LIN {X 0,Y 93.213,Z 295.861,A -85,B 0,C 180,E1 -28398.926,E2 -28398.926} C_VEL
LIN {X 0,Y 93.368,Z 291.962,A -85,B 0,C 180,E1 -28402.974,E2 -28402.974} C_VEL
LIN {X 0,Y 93.007,Z 287.711,A -85,B 0,C 180,E1 -28408.065,E2 -28408.065} C_VEL
LIN {X 0,Y 92.351,Z 284.316,A -85,B 0,C 180,E1 -28412.831,E2 -28412.831} C_VEL
LIN {X 0,Y 91.626,Z 281.752,A -85,B 0,C 180,E1 -28417.448,E2 -28417.448} C_VEL
LIN {X 0,Y 90.889,Z 279.975,A -85,B 0,C 180,E1 -28421.983,E2 -28421.983} C_VEL
LIN {X 0,Y 90.313,Z 278.726,A -85,B 0,C 180,E1 -28426.499,E2 -28426.499} C_VEL
LIN {X 0,Y 90.228,Z 277.226,A -85,B 0,C 180,E1 -28435.532,E2 -28435.532} C_VEL
LIN {X 0,Y 90.218,Z 278.004,A -85,B 0,C 180,E1 -28440,E2 -28440} C_VEL
LIN {X 0,Y 90.527,Z 282.078,A -85,B 0,C 180,E1 -28448.932,E2 -28448.932} C_VEL
LIN {X 0,Y 90.825,Z 283.273,A -85,B 0,C 180,E1 -28451.154,E2 -28451.154} C_VEL
LIN {X 0,Y 91.764,Z 288.136,A -85,B 0,C 180,E1 -28457.839,E2 -28457.839} C_VEL
LIN {X 0,Y 92.621,Z 293.238,A -85,B 0,C 180,E1 -28463.436,E2 -28463.436} C_VEL
LIN {X 0,Y 93.061,Z 299.729,A -85,B 0,C 180,E1 -28469.116,E2 -28469.116} C_VEL
LIN {X 0,Y 92.858,Z 301.798,A -85,B 0,C 180,E1 -28470.669,E2 -28470.669} C_VEL
LIN {X 0,Y 88.458,Z 309.904,A -85,B 0,C 180,E1 -28474.499,E2 -28474.499} C_VEL
LIN {X 0,Y 84.607,Z 315.889,A -85,B 0,C 180,E1 -28477.906,E2 -28477.906} C_VEL
LIN {X 0,Y 79.559,Z 323.019,A -85,B 0,C 180,E1 -28483.226,E2 -28483.226} C_VEL
LIN {X 0,Y 76.501,Z 327.119,A -85,B 0,C 180,E1 -28487.303,E2 -28487.303} C_VEL
LIN {X 0,Y 71.589,Z 332.386,A -85,B 0,C 180,E1 -28493.921,E2 -28493.921} C_VEL
LIN {X 0,Y 67.611,Z 336.755,A -85,B 0,C 180,E1 -28502.12,E2 -28502.12} C_VEL
LIN {X 0,Y 65.314,Z 339.861,A -85,B 0,C 180,E1 -28511.176,E2 -28511.176} C_VEL
LIN {X 0,Y 64.793,Z 341.313,A -85,B 0,C 180,E1 -28517.479,E2 -28517.479} C_VEL
LIN {X 0,Y 65.135,Z 342.235,A -85,B 0,C 180,E1 -28523.814,E2 -28523.814} C_VEL
LIN {X 0,Y 66.298,Z 342.706,A -85,B 0,C 180,E1 -28530.008,E2 -28530.008} C_VEL
LIN {X 0,Y 68.211,Z 342.64,A -85,B 0,C 180,E1 -28535.921,E2 -28535.921} C_VEL
LIN {X 0,Y 70.296,Z 342.047,A -85,B 0,C 180,E1 -28541.542,E2 -28541.542} C_VEL
LIN {X 0,Y 72.197,Z 340.793,A -85,B 0,C 180,E1 -28546.987,E2 -28546.987} C_VEL
LIN {X 0,Y 76.443,Z 338.002,A -85,B 0,C 180,E1 -28554.627,E2 -28554.627} C_VEL
LIN {X 0,Y 81.501,Z 346.039,A -85,B 0,C 180,E1 -28567.138,E2 -28567.138} C_VEL
LIN {X 0,Y 88.681,Z 351.555,A -85,B 0,C 180,E1 -28575.508,E2 -28575.508} C_VEL
LIN {X 0,Y 87.895,Z 350.817,A -85,B 0,C 180,E1 -28576.839,E2 -28576.839} C_VEL
LIN {X 0,Y 79.876,Z 342.499,A -85,B 0,C 180,E1 -28585.116,E2 -28585.116} C_VEL
LIN {X 0,Y 74.572,Z 333.187,A -85,B 0,C 180,E1 -28594.906,E2 -28594.906} C_VEL
LIN {X 0,Y 72.081,Z 324.848,A -85,B 0,C 180,E1 -28602.992,E2 -28602.992} C_VEL
LIN {X 0,Y 70.815,Z 316.559,A -85,B 0,C 180,E1 -28609.999,E2 -28609.999} C_VEL
LIN {X 0,Y 70.007,Z 307.489,A -85,B 0,C 180,E1 -28616.403,E2 -28616.403} C_VEL
LIN {X 0,Y 69.871,Z 305.556,A -85,B 0,C 180,E1 -28617.658,E2 -28617.658} C_VEL
LIN {X 0,Y 68.986,Z 305.923,A -85,B 0,C 180,E1 -28620,E2 -28620} C_VEL
LIN {X 0,Y 70.177,Z 304.044,A -85,B 0,C 180,E1 -28625.748,E2 -28625.748} C_VEL
LIN {X 0,Y 70.795,Z 303.378,A -85,B 0,C 180,E1 -28626.86,E2 -28626.86} C_VEL
LIN {X 0,Y 72.084,Z 302.243,A -85,B 0,C 180,E1 -28632.814,E2 -28632.814} C_VEL
LIN {X 0,Y 74.469,Z 300.381,A -85,B 0,C 180,E1 -28636.447,E2 -28636.447} C_VEL
LIN {X 0,Y 89.11,Z 292.891,A -85,B 0,C 180,E1 -28653.51,E2 -28653.51} C_VEL
LIN {X 0,Y 92.631,Z 292.592,A -85,B 0,C 180,E1 -28657.371,E2 -28657.371} C_VEL
LIN {X 0,Y 93.289,Z 293.19,A -85,B 0,C 180,E1 -28658.683,E2 -28658.683} C_VEL
LIN {X 0,Y 92.863,Z 296.646,A -85,B 0,C 180,E1 -28662.091,E2 -28662.091} C_VEL
LIN {X 0,Y 91.993,Z 299.53,A -85,B 0,C 180,E1 -28664.531,E2 -28664.531} C_VEL
LIN {X 0,Y 87.12,Z 305.638,A -85,B 0,C 180,E1 -28668.269,E2 -28668.269} C_VEL
LIN {X 0,Y 81.736,Z 311.304,A -85,B 0,C 180,E1 -28672.987,E2 -28672.987} C_VEL
LIN {X 0,Y 77.939,Z 314.962,A -85,B 0,C 180,E1 -28677.238,E2 -28677.238} C_VEL
LIN {X 0,Y 74.401,Z 318.347,A -85,B 0,C 180,E1 -28683.02,E2 -28683.02} C_VEL
LIN {X 0,Y 72.362,Z 319.71,A -85,B 0,C 180,E1 -28685.488,E2 -28685.488} C_VEL
LIN {X 0,Y 67.611,Z 321.736,A -85,B 0,C 180,E1 -28689.075,E2 -28689.075} C_VEL
LIN {X 0,Y 63.075,Z 323.435,A -85,B 0,C 180,E1 -28693.242,E2 -28693.242} C_VEL
LIN {X 0,Y 61.514,Z 324.146,A -85,B 0,C 180,E1 -28696.54,E2 -28696.54} C_VEL
LIN {X 0,Y 60.298,Z 324.937,A -85,B 0,C 180,E1 -28703.298,E2 -28703.298} C_VEL
LIN {X 0,Y 59.888,Z 325.215,A -85,B 0,C 180,E1 -28709.991,E2 -28709.991} C_VEL
LIN {X 0,Y 60.296,Z 324.966,A -85,B 0,C 180,E1 -28716.685,E2 -28716.685} C_VEL
LIN {X 0,Y 61.46,Z 324.257,A -85,B 0,C 180,E1 -28723.212,E2 -28723.212} C_VEL
LIN {X 0,Y 63.195,Z 323.047,A -85,B 0,C 180,E1 -28729.481,E2 -28729.481} C_VEL
LIN {X 0,Y 67.304,Z 320.204,A -85,B 0,C 180,E1 -28738.019,E2 -28738.019} C_VEL
LIN {X 0,Y 72.076,Z 316.138,A -85,B 0,C 180,E1 -28745.797,E2 -28745.797} C_VEL
LIN {X 0,Y 74.247,Z 314.396,A -85,B 0,C 180,E1 -28747.962,E2 -28747.962} C_VEL
LIN {X 0,Y 78.422,Z 310.454,A -85,B 0,C 180,E1 -28752.222,E2 -28752.222} C_VEL
LIN {X 0,Y 84.43,Z 304.214,A -85,B 0,C 180,E1 -28756.739,E2 -28756.739} C_VEL
LIN {X 0,Y 86.704,Z 301.543,A -85,B 0,C 180,E1 -28758.421,E2 -28758.421} C_VEL
LIN {X 0,Y 87.36,Z 299.906,A -85,B 0,C 180,E1 -28759.939,E2 -28759.939} C_VEL
LIN {X 0,Y 87.893,Z 297.12,A -85,B 0,C 180,E1 -28763.083,E2 -28763.083} C_VEL
LIN {X 0,Y 88.125,Z 294.71,A -85,B 0,C 180,E1 -28766.065,E2 -28766.065} C_VEL
LIN {X 0,Y 87.948,Z 290.964,A -85,B 0,C 180,E1 -28771.511,E2 -28771.511} C_VEL
LIN {X 0,Y 87.566,Z 288.203,A -85,B 0,C 180,E1 -28776.34,E2 -28776.34} C_VEL
LIN {X 0,Y 87.053,Z 286.287,A -85,B 0,C 180,E1 -28781.16,E2 -28781.16} C_VEL
LIN {X 0,Y 86.66,Z 284.824,A -85,B 0,C 180,E1 -28786.671,E2 -28786.671} C_VEL
LIN {X 0,Y 86.791,Z 283.5,A -85,B 0,C 180,E1 -28795.355,E2 -28795.355} C_VEL
LIN {X 0,Y 86.685,Z 284.411,A -85,B 0,C 180,E1 -28800,E2 -28800} C_VEL
LIN {X 0,Y 86.78,Z 288.516,A -85,B 0,C 180,E1 -28809.321,E2 -28809.321} C_VEL
LIN {X 0,Y 87.192,Z 293.1,A -85,B 0,C 180,E1 -28816.386,E2 -28816.386} C_VEL
LIN {X 0,Y 87.587,Z 296.996,A -85,B 0,C 180,E1 -28821.167,E2 -28821.167} C_VEL
LIN {X 0,Y 87.556,Z 301.883,A -85,B 0,C 180,E1 -28826.112,E2 -28826.112} C_VEL
LIN {X 0,Y 87.461,Z 303.785,A -85,B 0,C 180,E1 -28827.896,E2 -28827.896} C_VEL
LIN {X 0,Y 82.695,Z 311.486,A -85,B 0,C 180,E1 -28831.816,E2 -28831.816} C_VEL
LIN {X 0,Y 76.851,Z 319.303,A -85,B 0,C 180,E1 -28836.864,E2 -28836.864} C_VEL
LIN {X 0,Y 70.669,Z 326.788,A -85,B 0,C 180,E1 -28844.119,E2 -28844.119} C_VEL
LIN {X 0,Y 65.913,Z 331.38,A -85,B 0,C 180,E1 -28850.237,E2 -28850.237} C_VEL
LIN {X 0,Y 61.355,Z 335.759,A -85,B 0,C 180,E1 -28858.982,E2 -28858.982} C_VEL
LIN {X 0,Y 58.535,Z 338.861,A -85,B 0,C 180,E1 -28868.898,E2 -28868.898} C_VEL
LIN {X 0,Y 57.774,Z 340.433,A -85,B 0,C 180,E1 -28876.699,E2 -28876.699} C_VEL
LIN {X 0,Y 57.989,Z 341.238,A -85,B 0,C 180,E1 -28883.048,E2 -28883.048} C_VEL
LIN {X 0,Y 59.088,Z 341.706,A -85,B 0,C 180,E1 -28890.009,E2 -28890.009} C_VEL
LIN {X 0,Y 61.07,Z 341.644,A -85,B 0,C 180,E1 -28896.617,E2 -28896.617} C_VEL
LIN {X 0,Y 63.374,Z 341.065,A -85,B 0,C 180,E1 -28902.823,E2 -28902.823} C_VEL
LIN {X 0,Y 65.505,Z 339.817,A -85,B 0,C 180,E1 -28908.784,E2 -28908.784} C_VEL
LIN {X 0,Y 69.939,Z 337.021,A -85,B 0,C 180,E1 -28916.892,E2 -28916.892} C_VEL
LIN {X 0,Y 72.05,Z 335.766,A -85,B 0,C 180,E1 -28919.6,E2 -28919.6} C_VEL
LIN {X 0,Y 78.551,Z 343.736,A -85,B 0,C 180,E1 -28932.155,E2 -28932.155} C_VEL
LIN {X 0,Y 80.393,Z 345.2,A -85,B 0,C 180,E1 -28934.384,E2 -28934.384} C_VEL
LIN {X 0,Y 80.863,Z 345.457,A -85,B 0,C 180,E1 -28935.949,E2 -28935.949} C_VEL
LIN {X 0,Y 72.401,Z 335.446,A -85,B 0,C 180,E1 -28946.072,E2 -28946.072} C_VEL
LIN {X 0,Y 68.082,Z 326.403,A -85,B 0,C 180,E1 -28955.612,E2 -28955.612} C_VEL
LIN {X 0,Y 65.752,Z 317.359,A -85,B 0,C 180,E1 -28964.177,E2 -28964.177} C_VEL
LIN {X 0,Y 64.986,Z 312.689,A -85,B 0,C 180,E1 -28968.097,E2 -28968.097} C_VEL
LIN {X 0,Y 64.517,Z 312.846,A -85,B 0,C 180,E1 -28968.673,E2 -28968.673} C_VEL
LIN {X 0,Y 63.247,Z 312.343,A -85,B 0,C 180,E1 -28973.62,E2 -28973.62} C_VEL
LIN {X 0,Y 69.194,Z 305.675,A -85,B 0,C 180,E1 -28997.741,E2 -28997.741} C_VEL
LIN {X 0,Y 84.973,Z 298.241,A -85,B 0,C 180,E1 -29015.378,E2 -29015.378} C_VEL
LIN {X 0,Y 86.896,Z 297.908,A -85,B 0,C 180,E1 -29017.343,E2 -29017.343} C_VEL
LIN {X 0,Y 87.235,Z 299.689,A -85,B 0,C 180,E1 -29020.13,E2 -29020.13} C_VEL
LIN {X 0,Y 86.605,Z 301.357,A -85,B 0,C 180,E1 -29021.676,E2 -29021.676} C_VEL
LIN {X 0,Y 80.834,Z 307.865,A -85,B 0,C 180,E1 -29025.92,E2 -29025.92} C_VEL
LIN {X 0,Y 76.241,Z 312.297,A -85,B 0,C 180,E1 -29029.806,E2 -29029.806} C_VEL
LIN {X 0,Y 72.127,Z 315.945,A -85,B 0,C 180,E1 -29034.214,E2 -29034.214} C_VEL
LIN {X 0,Y 67.325,Z 320.057,A -85,B 0,C 180,E1 -29041.974,E2 -29041.974} C_VEL
LIN {X 0,Y 63.201,Z 322.96,A -85,B 0,C 180,E1 -29050.504,E2 -29050.504} C_VEL
LIN {X 0,Y 61.514,Z 324.146,A -85,B 0,C 180,E1 -29056.54,E2 -29056.54} C_VEL
LIN {X 0,Y 59.933,Z 325.036,A -85,B 0,C 180,E1 -29061.841,E2 -29061.841} C_VEL
LIN {X 0,Y 57.893,Z 325.631,A -85,B 0,C 180,E1 -29067.243,E2 -29067.243} C_VEL
LIN {X 0,Y 54.729,Z 325.742,A -85,B 0,C 180,E1 -29078.982,E2 -29078.982} C_VEL
LIN {X 0,Y 54.953,Z 325.039,A -85,B 0,C 180,E1 -29086.168,E2 -29086.168} C_VEL
LIN {X 0,Y 55.179,Z 324.847,A -85,B 0,C 180,E1 -29087.155,E2 -29087.155} C_VEL
LIN {X 0,Y 56.618,Z 324.02,A -85,B 0,C 180,E1 -29091.853,E2 -29091.853} C_VEL
LIN {X 0,Y 61.188,Z 321.181,A -85,B 0,C 180,E1 -29101.112,E2 -29101.112} C_VEL
LIN {X 0,Y 66.501,Z 317.119,A -85,B 0,C 180,E1 -29109.342,E2 -29109.342} C_VEL
LIN {X 0,Y 68.823,Z 315.385,A -85,B 0,C 180,E1 -29111.577,E2 -29111.577} C_VEL
LIN {X 0,Y 73.371,Z 311.451,A -85,B 0,C 180,E1 -29115.912,E2 -29115.912} C_VEL
LIN {X 0,Y 79.78,Z 305.234,A -85,B 0,C 180,E1 -29120.416,E2 -29120.416} C_VEL
LIN {X 0,Y 81.076,Z 303.837,A -85,B 0,C 180,E1 -29121.264,E2 -29121.264} C_VEL
LIN {X 0,Y 82.113,Z 302.004,A -85,B 0,C 180,E1 -29123.192,E2 -29123.192} C_VEL
LIN {X 0,Y 82.773,Z 298.468,A -85,B 0,C 180,E1 -29128.097,E2 -29128.097} C_VEL
LIN {X 0,Y 82.951,Z 296.421,A -85,B 0,C 180,E1 -29131.538,E2 -29131.538} C_VEL
LIN {X 0,Y 82.981,Z 294.488,A -85,B 0,C 180,E1 -29134.946,E2 -29134.946} C_VEL
LIN {X 0,Y 82.785,Z 292.446,A -85,B 0,C 180,E1 -29140.149,E2 -29140.149} C_VEL
LIN {X 0,Y 82.557,Z 291.033,A -85,B 0,C 180,E1 -29145.203,E2 -29145.203} C_VEL
LIN {X 0,Y 82.524,Z 290.077,A -85,B 0,C 180,E1 -29150.193,E2 -29150.193} C_VEL
LIN {X 0,Y 82.86,Z 289.48,A -85,B 0,C 180,E1 -29155.134,E2 -29155.134} C_VEL
LIN {X 0,Y 82.631,Z 290.523,A -85,B 0,C 180,E1 -29160,E2 -29160} C_VEL
LIN {X 0,Y 82.398,Z 293.511,A -85,B 0,C 180,E1 -29167.35,E2 -29167.35} C_VEL
LIN {X 0,Y 82.465,Z 297.897,A -85,B 0,C 180,E1 -29174.813,E2 -29174.813} C_VEL
LIN {X 0,Y 82.414,Z 301.877,A -85,B 0,C 180,E1 -29180.295,E2 -29180.295} C_VEL
LIN {X 0,Y 82.123,Z 305.246,A -85,B 0,C 180,E1 -29183.984,E2 -29183.984} C_VEL
LIN {X 0,Y 81.822,Z 306.439,A -85,B 0,C 180,E1 -29185.093,E2 -29185.093} C_VEL
LIN {X 0,Y 76.479,Z 313.761,A -85,B 0,C 180,E1 -29189.206,E2 -29189.206} C_VEL
LIN {X 0,Y 70.288,Z 320.909,A -85,B 0,C 180,E1 -29194.435,E2 -29194.435} C_VEL
LIN {X 0,Y 64.858,Z 326.701,A -85,B 0,C 180,E1 -29200.68,E2 -29200.68} C_VEL
LIN {X 0,Y 58.648,Z 331.979,A -85,B 0,C 180,E1 -29208.782,E2 -29208.782} C_VEL
LIN {X 0,Y 53.957,Z 335.938,A -85,B 0,C 180,E1 -29218.612,E2 -29218.612} C_VEL
LIN {X 0,Y 51.876,Z 337.862,A -85,B 0,C 180,E1 -29226.03,E2 -29226.03} C_VEL
LIN {X 0,Y 50.745,Z 339.56,A -85,B 0,C 180,E1 -29235.808,E2 -29235.808} C_VEL
LIN {X 0,Y 51.882,Z 340.708,A -85,B 0,C 180,E1 -29250.01,E2 -29250.01} C_VEL
LIN {X 0,Y 53.933,Z 340.648,A -85,B 0,C 180,E1 -29257.497,E2 -29257.497} C_VEL
LIN {X 0,Y 56.488,Z 340.083,A -85,B 0,C 180,E1 -29264.418,E2 -29264.418} C_VEL
LIN {X 0,Y 58.891,Z 338.842,A -85,B 0,C 180,E1 -29270.988,E2 -29270.988} C_VEL
LIN {X 0,Y 63.758,Z 336.045,A -85,B 0,C 180,E1 -29279.747,E2 -29279.747} C_VEL
LIN {X 0,Y 68.349,Z 333.34,A -85,B 0,C 180,E1 -29285.121,E2 -29285.121} C_VEL
LIN {X 0,Y 72.467,Z 338.121,A -85,B 0,C 180,E1 -29292.765,E2 -29292.765} C_VEL
LIN {X 0,Y 73.474,Z 338.931,A -85,B 0,C 180,E1 -29295.492,E2 -29295.492} C_VEL
LIN {X 0,Y 65.909,Z 328.893,A -85,B 0,C 180,E1 -29305.957,E2 -29305.957} C_VEL
LIN {X 0,Y 61.913,Z 319.719,A -85,B 0,C 180,E1 -29315.703,E2 -29315.703} C_VEL
LIN {X 0,Y 59.726,Z 319.453,A -85,B 0,C 180,E1 -29319.329,E2 -29319.329} C_VEL
LIN {X 0,Y 58.865,Z 318.697,A -85,B 0,C 180,E1 -29322.8,E2 -29322.8} C_VEL
LIN {X 0,Y 58.688,Z 317.695,A -85,B 0,C 180,E1 -29326.143,E2 -29326.143} C_VEL
LIN {X 0,Y 57.591,Z 316.558,A -85,B 0,C 180,E1 -29332.991,E2 -29332.991} C_VEL
LIN {X 0,Y 64.059,Z 310.157,A -85,B 0,C 180,E1 -29359.704,E2 -29359.704} C_VEL
LIN {X 0,Y 80.664,Z 303.228,A -85,B 0,C 180,E1 -29377.582,E2 -29377.582} C_VEL
LIN {X 0,Y 81.128,Z 303.553,A -85,B 0,C 180,E1 -29378.761,E2 -29378.761} C_VEL
LIN {X 0,Y 74.651,Z 310.085,A -85,B 0,C 180,E1 -29383.136,E2 -29383.136} C_VEL
LIN {X 0,Y 68.822,Z 315.179,A -85,B 0,C 180,E1 -29388.402,E2 -29388.402} C_VEL
LIN {X 0,Y 64.64,Z 318.465,A -85,B 0,C 180,E1 -29393.264,E2 -29393.264} C_VEL
LIN {X 0,Y 59.567,Z 322.125,A -85,B 0,C 180,E1 -29401.83,E2 -29401.83} C_VEL
LIN {X 0,Y 56.625,Z 323.933,A -85,B 0,C 180,E1 -29408.13,E2 -29408.13} C_VEL
LIN {X 0,Y 54.646,Z 325.166,A -85,B 0,C 180,E1 -29415.085,E2 -29415.085} C_VEL
LIN {X 0,Y 53.324,Z 325.911,A -85,B 0,C 180,E1 -29422.417,E2 -29422.417} C_VEL
LIN {X 0,Y 52.86,Z 326.189,A -85,B 0,C 180,E1 -29429.99,E2 -29429.99} C_VEL
LIN {X 0,Y 53.322,Z 325.94,A -85,B 0,C 180,E1 -29437.564,E2 -29437.564} C_VEL
LIN {X 0,Y 55.179,Z 324.847,A -85,B 0,C 180,E1 -29447.155,E2 -29447.155} C_VEL
LIN {X 0,Y 55.721,Z 324.302,A -85,B 0,C 180,E1 -29451.189,E2 -29451.189} C_VEL
LIN {X 0,Y 55.563,Z 323.295,A -85,B 0,C 180,E1 -29458.062,E2 -29458.062} C_VEL
LIN {X 0,Y 56.037,Z 321.967,A -85,B 0,C 180,E1 -29464.849,E2 -29464.849} C_VEL
LIN {X 0,Y 57.47,Z 320.74,A -85,B 0,C 180,E1 -29468.41,E2 -29468.41} C_VEL
LIN {X 0,Y 61.226,Z 318.1,A -85,B 0,C 180,E1 -29473.517,E2 -29473.517} C_VEL
LIN {X 0,Y 66.062,Z 314.523,A -85,B 0,C 180,E1 -29478.121,E2 -29478.121} C_VEL
LIN {X 0,Y 72.735,Z 308.945,A -85,B 0,C 180,E1 -29482.847,E2 -29482.847} C_VEL
LIN {X 0,Y 76.073,Z 305.67,A -85,B 0,C 180,E1 -29484.875,E2 -29484.875} C_VEL
LIN {X 0,Y 76.573,Z 304.932,A -85,B 0,C 180,E1 -29485.68,E2 -29485.68} C_VEL
LIN {X 0,Y 77.416,Z 302.319,A -85,B 0,C 180,E1 -29490.046,E2 -29490.046} C_VEL
LIN {X 0,Y 77.81,Z 300.007,A -85,B 0,C 180,E1 -29494.569,E2 -29494.569} C_VEL
LIN {X 0,Y 78.036,Z 298.307,A -85,B 0,C 180,E1 -29498.885,E2 -29498.885} C_VEL
LIN {X 0,Y 77.964,Z 296.797,A -85,B 0,C 180,E1 -29504.31,E2 -29504.31} C_VEL
LIN {X 0,Y 78.216,Z 295.608,A -85,B 0,C 180,E1 -29511.213,E2 -29511.213} C_VEL
LIN {X 0,Y 78.576,Z 295.249,A -85,B 0,C 180,E1 -29514.868,E2 -29514.868} C_VEL
LIN {X 0,Y 78.21,Z 296.396,A -85,B 0,C 180,E1 -29520,E2 -29520} C_VEL
LIN {X 0,Y 77.687,Z 299.36,A -85,B 0,C 180,E1 -29527.537,E2 -29527.537} C_VEL
LIN {X 0,Y 77.446,Z 302.348,A -85,B 0,C 180,E1 -29533.113,E2 -29533.113} C_VEL
LIN {X 0,Y 77.367,Z 304.022,A -85,B 0,C 180,E1 -29535.814,E2 -29535.814} C_VEL
LIN {X 0,Y 76.875,Z 307.048,A -85,B 0,C 180,E1 -29540.081,E2 -29540.081} C_VEL
LIN {X 0,Y 76.609,Z 308.213,A -85,B 0,C 180,E1 -29541.528,E2 -29541.528} C_VEL
LIN {X 0,Y 71.783,Z 314.191,A -85,B 0,C 180,E1 -29545.11,E2 -29545.11} C_VEL
LIN {X 0,Y 65.12,Z 321.119,A -85,B 0,C 180,E1 -29550.318,E2 -29550.318} C_VEL
LIN {X 0,Y 59.75,Z 326.157,A -85,B 0,C 180,E1 -29556.023,E2 -29556.023} C_VEL
LIN {X 0,Y 53.458,Z 330.98,A -85,B 0,C 180,E1 -29563.706,E2 -29563.706} C_VEL
LIN {X 0,Y 47.964,Z 334.939,A -85,B 0,C 180,E1 -29574.132,E2 -29574.132} C_VEL
LIN {X 0,Y 45.409,Z 336.867,A -85,B 0,C 180,E1 -29582.347,E2 -29582.347} C_VEL
LIN {X 0,Y 43.719,Z 338.691,A -85,B 0,C 180,E1 -29594.691,E2 -29594.691} C_VEL
LIN {X 0,Y 44.681,Z 339.709,A -85,B 0,C 180,E1 -29610.012,E2 -29610.012} C_VEL
LIN {X 0,Y 46.806,Z 339.651,A -85,B 0,C 180,E1 -29618.647,E2 -29618.647} C_VEL
LIN {X 0,Y 49.625,Z 339.095,A -85,B 0,C 180,E1 -29626.465,E2 -29626.465} C_VEL
LIN {X 0,Y 52.385,Z 337.867,A -85,B 0,C 180,E1 -29633.744,E2 -29633.744} C_VEL
LIN {X 0,Y 57.78,Z 335.071,A -85,B 0,C 180,E1 -29643.196,E2 -29643.196} C_VEL
LIN {X 0,Y 64.957,Z 330.914,A -85,B 0,C 180,E1 -29650.768,E2 -29650.768} C_VEL
LIN {X 0,Y 65.352,Z 330.748,A -85,B 0,C 180,E1 -29650.978,E2 -29650.978} C_VEL
LIN {X 0,Y 66.65,Z 332.128,A -85,B 0,C 180,E1 -29653.278,E2 -29653.278} C_VEL
LIN {X 0,Y 65.7,Z 330.947,A -85,B 0,C 180,E1 -29655.948,E2 -29655.948} C_VEL
LIN {X 0,Y 62.341,Z 326.675,A -85,B 0,C 180,E1 -29660.644,E2 -29660.644} C_VEL
LIN {X 0,Y 59.478,Z 326.17,A -85,B 0,C 180,E1 -29663.786,E2 -29663.786} C_VEL
LIN {X 0,Y 56.368,Z 324.425,A -85,B 0,C 180,E1 -29670.8,E2 -29670.8} C_VEL
LIN {X 0,Y 55.253,Z 316.008,A -85,B 0,C 180,E1 -29714.738,E2 -29714.738} C_VEL
LIN {X 0,Y 71.112,Z 309.429,A -85,B 0,C 180,E1 -29736.37,E2 -29736.37} C_VEL
LIN {X 0,Y 71.406,Z 309.881,A -85,B 0,C 180,E1 -29738.047,E2 -29738.047} C_VEL
LIN {X 0,Y 66.127,Z 314.281,A -85,B 0,C 180,E1 -29741.919,E2 -29741.919} C_VEL
LIN {X 0,Y 61.275,Z 317.911,A -85,B 0,C 180,E1 -29746.503,E2 -29746.503} C_VEL
LIN {X 0,Y 55.312,Z 322.016,A -85,B 0,C 180,E1 -29755.115,E2 -29755.115} C_VEL
LIN {X 0,Y 50.171,Z 324.907,A -85,B 0,C 180,E1 -29765.139,E2 -29765.139} C_VEL
LIN {X 0,Y 47.889,Z 326.141,A -85,B 0,C 180,E1 -29772.921,E2 -29772.921} C_VEL
LIN {X 0,Y 46.367,Z 326.885,A -85,B 0,C 180,E1 -29781.271,E2 -29781.271} C_VEL
LIN {X 0,Y 45.832,Z 327.163,A -85,B 0,C 180,E1 -29789.989,E2 -29789.989} C_VEL
LIN {X 0,Y 46.364,Z 326.914,A -85,B 0,C 180,E1 -29798.707,E2 -29798.707} C_VEL
LIN {X 0,Y 48.483,Z 325.835,A -85,B 0,C 180,E1 -29809.509,E2 -29809.509} C_VEL
LIN {X 0,Y 50.163,Z 324.993,A -85,B 0,C 180,E1 -29814.842,E2 -29814.842} C_VEL
LIN {X 0,Y 55.29,Z 322.159,A -85,B 0,C 180,E1 -29824.878,E2 -29824.878} C_VEL
LIN {X 0,Y 57.47,Z 320.74,A -85,B 0,C 180,E1 -29828.41,E2 -29828.41} C_VEL
LIN {X 0,Y 61.484,Z 317.785,A -85,B 0,C 180,E1 -29834.343,E2 -29834.343} C_VEL
LIN {X 0,Y 65.334,Z 314.38,A -85,B 0,C 180,E1 -29839.825,E2 -29839.825} C_VEL
LIN {X 0,Y 68.751,Z 310.719,A -85,B 0,C 180,E1 -29845.067,E2 -29845.067} C_VEL
LIN {X 0,Y 71.486,Z 306.974,A -85,B 0,C 180,E1 -29850.321,E2 -29850.321} C_VEL
LIN {X 0,Y 72.401,Z 304.927,A -85,B 0,C 180,E1 -29854.663,E2 -29854.663} C_VEL
LIN {X 0,Y 72.629,Z 303.994,A -85,B 0,C 180,E1 -29857.228,E2 -29857.228} C_VEL
LIN {X 0,Y 73.012,Z 302.032,A -85,B 0,C 180,E1 -29864.249,E2 -29864.249} C_VEL
LIN {X 0,Y 73.275,Z 301.298,A -85,B 0,C 180,E1 -29868.94,E2 -29868.94} C_VEL
LIN {X 0,Y 73.895,Z 300.693,A -85,B 0,C 180,E1 -29874.542,E2 -29874.542} C_VEL
LIN {X 0,Y 73.398,Z 301.932,A -85,B 0,C 180,E1 -29880,E2 -29880} C_VEL
LIN {X 0,Y 72.847,Z 303.865,A -85,B 0,C 180,E1 -29885.536,E2 -29885.536} C_VEL
LIN {X 0,Y 72.067,Z 307.371,A -85,B 0,C 180,E1 -29892.822,E2 -29892.822} C_VEL
LIN {X 0,Y 71.519,Z 310,A -85,B 0,C 180,E1 -29897.145,E2 -29897.145} C_VEL
LIN {X 0,Y 70.098,Z 311.932,A -85,B 0,C 180,E1 -29898.766,E2 -29898.766} C_VEL
LIN {X 0,Y 63.144,Z 318.804,A -85,B 0,C 180,E1 -29903.352,E2 -29903.352} C_VEL
LIN {X 0,Y 56.371,Z 324.624,A -85,B 0,C 180,E1 -29909.244,E2 -29909.244} C_VEL
LIN {X 0,Y 51.242,Z 328.37,A -85,B 0,C 180,E1 -29914.64,E2 -29914.64} C_VEL
LIN {X 0,Y 44.301,Z 332.77,A -85,B 0,C 180,E1 -29924.465,E2 -29924.465} C_VEL
LIN {X 0,Y 39.174,Z 335.87,A -85,B 0,C 180,E1 -29937.454,E2 -29937.454} C_VEL
LIN {X 0,Y 36.726,Z 337.818,A -85,B 0,C 180,E1 -29953.097,E2 -29953.097} C_VEL
LIN {X 0,Y 37.479,Z 338.711,A -85,B 0,C 180,E1 -29970.014,E2 -29970.014} C_VEL
LIN {X 0,Y 39.72,Z 338.655,A -85,B 0,C 180,E1 -29980.205,E2 -29980.205} C_VEL
LIN {X 0,Y 42.848,Z 338.108,A -85,B 0,C 180,E1 -29989.163,E2 -29989.163} C_VEL
LIN {X 0,Y 46.033,Z 336.891,A -85,B 0,C 180,E1 -29997.272,E2 -29997.272} C_VEL
LIN {X 0,Y 52.054,Z 334.096,A -85,B 0,C 180,E1 -30007.426,E2 -30007.426} C_VEL
LIN {X 0,Y 58.466,Z 330.668,A -85,B 0,C 180,E1 -30014.184,E2 -30014.184} C_VEL
LIN {X 0,Y 56.737,Z 329.725,A -85,B 0,C 180,E1 -30017.351,E2 -30017.351} C_VEL
LIN {X 0,Y 54.477,Z 329.309,A -85,B 0,C 180,E1 -30019.831,E2 -30019.831} C_VEL
LIN {X 0,Y 46.456,Z 325.121,A -85,B 0,C 180,E1 -30042.389,E2 -30042.389} C_VEL
LIN {X 0,Y 49.245,Z 319.665,A -85,B 0,C 180,E1 -30076.585,E2 -30076.585} C_VEL
LIN {X 0,Y 61.249,Z 315.012,A -85,B 0,C 180,E1 -30095.011,E2 -30095.011} C_VEL
LIN {X 0,Y 61.659,Z 315.273,A -85,B 0,C 180,E1 -30097.06,E2 -30097.06} C_VEL
LIN {X 0,Y 56.382,Z 318.893,A -85,B 0,C 180,E1 -30101.579,E2 -30101.579} C_VEL
LIN {X 0,Y 49.709,Z 322.996,A -85,B 0,C 180,E1 -30110.477,E2 -30110.477} C_VEL
LIN {X 0,Y 43.894,Z 325.881,A -85,B 0,C 180,E1 -30121.279,E2 -30121.279} C_VEL
LIN {X 0,Y 41.223,Z 327.116,A -85,B 0,C 180,E1 -30130.051,E2 -30130.051} C_VEL
LIN {X 0,Y 39.435,Z 327.858,A -85,B 0,C 180,E1 -30139.721,E2 -30139.721} C_VEL
LIN {X 0,Y 38.804,Z 328.138,A -85,B 0,C 180,E1 -30149.987,E2 -30149.987} C_VEL
LIN {X 0,Y 39.432,Z 327.888,A -85,B 0,C 180,E1 -30160.253,E2 -30160.253} C_VEL
LIN {X 0,Y 41.217,Z 327.179,A -85,B 0,C 180,E1 -30169.926,E2 -30169.926} C_VEL
LIN {X 0,Y 43.885,Z 325.965,A -85,B 0,C 180,E1 -30178.7,E2 -30178.7} C_VEL
LIN {X 0,Y 49.686,Z 323.136,A -85,B 0,C 180,E1 -30189.518,E2 -30189.518} C_VEL
LIN {X 0,Y 56.336,Z 319.081,A -85,B 0,C 180,E1 -30198.447,E2 -30198.447} C_VEL
LIN {X 0,Y 62.965,Z 314.518,A -85,B 0,C 180,E1 -30204.006,E2 -30204.006} C_VEL
LIN {X 0,Y 70.81,Z 308.071,A -85,B 0,C 180,E1 -30208.671,E2 -30208.671} C_VEL
LIN {X 0,Y 71.486,Z 306.974,A -85,B 0,C 180,E1 -30210.321,E2 -30210.321} C_VEL
LIN {X 0,Y 71.789,Z 305.981,A -85,B 0,C 180,E1 -30212.685,E2 -30212.685} C_VEL
LIN {X 0,Y 71.259,Z 305.686,A -85,B 0,C 180,E1 -30215.235,E2 -30215.235} C_VEL
LIN {X 0,Y 70.099,Z 305.903,A -85,B 0,C 180,E1 -30218.332,E2 -30218.332} C_VEL
LIN {X 0,Y 67.937,Z 306.699,A -85,B 0,C 180,E1 -30225.257,E2 -30225.257} C_VEL
LIN {X 0,Y 67.991,Z 306.489,A -85,B 0,C 180,E1 -30227.647,E2 -30227.647} C_VEL
LIN {X 0,Y 68.727,Z 305.783,A -85,B 0,C 180,E1 -30234.13,E2 -30234.13} C_VEL
LIN {X 0,Y 68.125,Z 307.065,A -85,B 0,C 180,E1 -30240,E2 -30240} C_VEL
LIN {X 0,Y 67.326,Z 309.188,A -85,B 0,C 180,E1 -30245.992,E2 -30245.992} C_VEL
LIN {X 0,Y 66.383,Z 311.911,A -85,B 0,C 180,E1 -30252.224,E2 -30252.224} C_VEL
LIN {X 0,Y 65.281,Z 313.544,A -85,B 0,C 180,E1 -30254.357,E2 -30254.357} C_VEL
LIN {X 0,Y 57.566,Z 320.229,A -85,B 0,C 180,E1 -30258.917,E2 -30258.917} C_VEL
LIN {X 0,Y 50.547,Z 325.425,A -85,B 0,C 180,E1 -30264.652,E2 -30264.652} C_VEL
LIN {X 0,Y 42.095,Z 330.444,A -85,B 0,C 180,E1 -30273.43,E2 -30273.43} C_VEL
LIN {X 0,Y 37.265,Z 332.939,A -85,B 0,C 180,E1 -30281.051,E2 -30281.051} C_VEL
LIN {X 0,Y 33.344,Z 334.876,A -85,B 0,C 180,E1 -30290.8,E2 -30290.8} C_VEL
LIN {X 0,Y 29.781,Z 336.941,A -85,B 0,C 180,E1 -30310.727,E2 -30310.727} C_VEL
LIN {X 0,Y 30.271,Z 337.712,A -85,B 0,C 180,E1 -30330.017,E2 -30330.017} C_VEL
LIN {X 0,Y 32.665,Z 337.657,A -85,B 0,C 180,E1 -30342.441,E2 -30342.441} C_VEL
LIN {X 0,Y 36.18,Z 337.117,A -85,B 0,C 180,E1 -30352.877,E2 -30352.877} C_VEL
LIN {X 0,Y 39.909,Z 335.914,A -85,B 0,C 180,E1 -30361.906,E2 -30361.906} C_VEL
LIN {X 0,Y 46.677,Z 333.119,A -85,B 0,C 180,E1 -30372.668,E2 -30372.668} C_VEL
LIN {X 0,Y 48.75,Z 331.795,A -85,B 0,C 180,E1 -30376.137,E2 -30376.137} C_VEL
LIN {X 0,Y 40.229,Z 328.042,A -85,B 0,C 180,E1 -30399.55,E2 -30399.55} C_VEL
LIN {X 0,Y 43.079,Z 322.832,A -85,B 0,C 180,E1 -30439.044,E2 -30439.044} C_VEL
LIN {X 0,Y 51.1,Z 319.97,A -85,B 0,C 180,E1 -30453.377,E2 -30453.377} C_VEL
LIN {X 0,Y 51.994,Z 319.874,A -85,B 0,C 180,E1 -30455.789,E2 -30455.789} C_VEL
LIN {X 0,Y 44.513,Z 323.976,A -85,B 0,C 180,E1 -30464.709,E2 -30464.709} C_VEL
LIN {X 0,Y 37.882,Z 326.854,A -85,B 0,C 180,E1 -30476.165,E2 -30476.165} C_VEL
LIN {X 0,Y 34.7,Z 328.091,A -85,B 0,C 180,E1 -30486.088,E2 -30486.088} C_VEL
LIN {X 0,Y 32.544,Z 328.832,A -85,B 0,C 180,E1 -30497.512,E2 -30497.512} C_VEL
LIN {X 0,Y 31.776,Z 329.112,A -85,B 0,C 180,E1 -30509.984,E2 -30509.984} C_VEL
LIN {X 0,Y 32.54,Z 328.861,A -85,B 0,C 180,E1 -30522.457,E2 -30522.457} C_VEL
LIN {X 0,Y 34.692,Z 328.153,A -85,B 0,C 180,E1 -30533.885,E2 -30533.885} C_VEL
LIN {X 0,Y 37.871,Z 326.938,A -85,B 0,C 180,E1 -30543.813,E2 -30543.813} C_VEL
LIN {X 0,Y 44.489,Z 324.114,A -85,B 0,C 180,E1 -30555.288,E2 -30555.288} C_VEL
LIN {X 0,Y 51.939,Z 320.062,A -85,B 0,C 180,E1 -30564.262,E2 -30564.262} C_VEL
LIN {X 0,Y 60.625,Z 314.442,A -85,B 0,C 180,E1 -30570.375,E2 -30570.375} C_VEL
LIN {X 0,Y 65.689,Z 310.578,A -85,B 0,C 180,E1 -30572.957,E2 -30572.957} C_VEL
LIN {X 0,Y 66.608,Z 309.416,A -85,B 0,C 180,E1 -30575.036,E2 -30575.036} C_VEL
LIN {X 0,Y 67.421,Z 307.49,A -85,B 0,C 180,E1 -30581.776,E2 -30581.776} C_VEL
LIN {X 0,Y 67.991,Z 306.489,A -85,B 0,C 180,E1 -30587.647,E2 -30587.647} C_VEL
LIN {X 0,Y 67.897,Z 306.527,A -85,B 0,C 180,E1 -30590.316,E2 -30590.316} C_VEL
LIN {X 0,Y 66.648,Z 307.714,A -85,B 0,C 180,E1 -30593.916,E2 -30593.916} C_VEL
LIN {X 0,Y 61.954,Z 312.861,A -85,B 0,C 180,E1 -30603.429,E2 -30603.429} C_VEL
LIN {X 0,Y 61.676,Z 313.348,A -85,B 0,C 180,E1 -30604.654,E2 -30604.654} C_VEL
LIN {X 0,Y 61.369,Z 314.051,A -85,B 0,C 180,E1 -30606.576,E2 -30606.576} C_VEL
LIN {X 0,Y 60.224,Z 315.658,A -85,B 0,C 180,E1 -30609.559,E2 -30609.559} C_VEL
LIN {X 0,Y 50.825,Z 322.545,A -85,B 0,C 180,E1 -30614.588,E2 -30614.588} C_VEL
LIN {X 0,Y 44.641,Z 326.351,A -85,B 0,C 180,E1 -30619.196,E2 -30619.196} C_VEL
LIN {X 0,Y 35.728,Z 330.773,A -85,B 0,C 180,E1 -30627.756,E2 -30627.756} C_VEL
LIN {X 0,Y 28.134,Z 333.879,A -85,B 0,C 180,E1 -30641.49,E2 -30641.49} C_VEL
LIN {X 0,Y 22.968,Z 336.036,A -85,B 0,C 180,E1 -30666.629,E2 -30666.629} C_VEL
LIN {X 0,Y 23.071,Z 336.714,A -85,B 0,C 180,E1 -30690.023,E2 -30690.023} C_VEL
LIN {X 0,Y 25.669,Z 336.657,A -85,B 0,C 180,E1 -30705.911,E2 -30705.911} C_VEL
LIN {X 0,Y 29.739,Z 336.128,A -85,B 0,C 180,E1 -30718.226,E2 -30718.226} C_VEL
LIN {X 0,Y 34.134,Z 334.936,A -85,B 0,C 180,E1 -30728.165,E2 -30728.165} C_VEL
LIN {X 0,Y 39.097,Z 333.207,A -85,B 0,C 180,E1 -30735.994,E2 -30735.994} C_VEL
LIN {X 0,Y 36.693,Z 331.775,A -85,B 0,C 180,E1 -30744.929,E2 -30744.929} C_VEL
LIN {X 0,Y 42.579,Z 323.749,A -85,B 0,C 180,E1 -30814.361,E2 -30814.361} C_VEL
LIN {X 0,Y 37.23,Z 326.035,A -85,B 0,C 180,E1 -30820.946,E2 -30820.946} C_VEL
LIN {X 0,Y 32.282,Z 327.828,A -85,B 0,C 180,E1 -30829.202,E2 -30829.202} C_VEL
LIN {X 0,Y 28.418,Z 329.066,A -85,B 0,C 180,E1 -30840.335,E2 -30840.335} C_VEL
LIN {X 0,Y 25.727,Z 329.807,A -85,B 0,C 180,E1 -30854.126,E2 -30854.126} C_VEL
LIN {X 0,Y 24.748,Z 330.086,A -85,B 0,C 180,E1 -30869.979,E2 -30869.979} C_VEL
LIN {X 0,Y 25.722,Z 329.834,A -85,B 0,C 180,E1 -30885.835,E2 -30885.835} C_VEL
LIN {X 0,Y 28.409,Z 329.127,A -85,B 0,C 180,E1 -30899.634,E2 -30899.634} C_VEL
LIN {X 0,Y 32.27,Z 327.911,A -85,B 0,C 180,E1 -30910.774,E2 -30910.774} C_VEL
LIN {X 0,Y 39.859,Z 325.091,A -85,B 0,C 180,E1 -30922.488,E2 -30922.488} C_VEL
LIN {X 0,Y 48.172,Z 321.043,A -85,B 0,C 180,E1 -30931.066,E2 -30931.066} C_VEL
LIN {X 0,Y 57.477,Z 315.439,A -85,B 0,C 180,E1 -30936.476,E2 -30936.476} C_VEL
LIN {X 0,Y 60.711,Z 313.174,A -85,B 0,C 180,E1 -30937.809,E2 -30937.809} C_VEL
LIN {X 0,Y 61.37,Z 312.444,A -85,B 0,C 180,E1 -30939.906,E2 -30939.906} C_VEL
LIN {X 0,Y 62.437,Z 311.049,A -85,B 0,C 180,E1 -30948.402,E2 -30948.402} C_VEL
LIN {X 0,Y 63.195,Z 310.526,A -85,B 0,C 180,E1 -30953.615,E2 -30953.615} C_VEL
LIN {X 0,Y 62.508,Z 311.785,A -85,B 0,C 180,E1 -30960,E2 -30960} C_VEL
LIN {X 0,Y 61.676,Z 313.348,A -85,B 0,C 180,E1 -30964.654,E2 -30964.654} C_VEL
LIN {X 0,Y 60.723,Z 314.497,A -85,B 0,C 180,E1 -30966.382,E2 -30966.382} C_VEL
LIN {X 0,Y 58.578,Z 316.288,A -85,B 0,C 180,E1 -30967.664,E2 -30967.664} C_VEL
LIN {X 0,Y 54.781,Z 318.852,A -85,B 0,C 180,E1 -30968.261,E2 -30968.261} C_VEL
LIN {X 0,Y 46.706,Z 323.29,A -85,B 0,C 180,E1 -30968.264,E2 -30968.264} C_VEL
LIN {X 0,Y 44.095,Z 324.648,A -85,B 0,C 180,E1 -30969.175,E2 -30969.175} C_VEL
LIN {X 0,Y 36.22,Z 328.448,A -85,B 0,C 180,E1 -30974.086,E2 -30974.086} C_VEL
LIN {X 0,Y 29.857,Z 330.941,A -85,B 0,C 180,E1 -30979.737,E2 -30979.737} C_VEL
LIN {X 0,Y 23.987,Z 332.884,A -85,B 0,C 180,E1 -30988.526,E2 -30988.526} C_VEL
LIN {X 0,Y 19.044,Z 334.331,A -85,B 0,C 180,E1 -31002.473,E2 -31002.473} C_VEL
LIN {X 0,Y 15.945,Z 335.247,A -85,B 0,C 180,E1 -31023.884,E2 -31023.884} C_VEL
LIN {X 0,Y 15.877,Z 335.717,A -85,B 0,C 180,E1 -31050.033,E2 -31050.033} C_VEL
LIN {X 0,Y 18.85,Z 335.659,A -85,B 0,C 180,E1 -31071.92,E2 -31071.92} C_VEL
LIN {X 0,Y 23.668,Z 335.134,A -85,B 0,C 180,E1 -31086.46,E2 -31086.46} C_VEL
LIN {X 0,Y 28.924,Z 333.96,A -85,B 0,C 180,E1 -31096.824,E2 -31096.824} C_VEL
LIN {X 0,Y 29.791,Z 333.228,A -85,B 0,C 180,E1 -31101.961,E2 -31101.961} C_VEL
LIN {X 0,Y 31.611,Z 327.453,A -85,B 0,C 180,E1 -31169.838,E2 -31169.838} C_VEL
LIN {X 0,Y 29.767,Z 328.086,A -85,B 0,C 180,E1 -31175.77,E2 -31175.77} C_VEL
LIN {X 0,Y 22.581,Z 330.041,A -85,B 0,C 180,E1 -31191.474,E2 -31191.474} C_VEL
LIN {X 0,Y 19.064,Z 330.781,A -85,B 0,C 180,E1 -31208.339,E2 -31208.339} C_VEL
LIN {X 0,Y 17.72,Z 331.06,A -85,B 0,C 180,E1 -31229.971,E2 -31229.971} C_VEL
LIN {X 0,Y 19.057,Z 330.808,A -85,B 0,C 180,E1 -31251.611,E2 -31251.611} C_VEL
LIN {X 0,Y 22.569,Z 330.101,A -85,B 0,C 180,E1 -31268.491,E2 -31268.491} C_VEL
LIN {X 0,Y 27.336,Z 328.884,A -85,B 0,C 180,E1 -31280.44,E2 -31280.44} C_VEL
LIN {X 0,Y 36.013,Z 326.068,A -85,B 0,C 180,E1 -31291.394,E2 -31291.394} C_VEL
LIN {X 0,Y 45.191,Z 322.024,A -85,B 0,C 180,E1 -31298.892,E2 -31298.892} C_VEL
LIN {X 0,Y 55.066,Z 316.425,A -85,B 0,C 180,E1 -31303.204,E2 -31303.204} C_VEL
LIN {X 0,Y 56.107,Z 315.672,A -85,B 0,C 180,E1 -31305.491,E2 -31305.491} C_VEL
LIN {X 0,Y 57.336,Z 314.966,A -85,B 0,C 180,E1 -31312.959,E2 -31312.959} C_VEL
LIN {X 0,Y 56.526,Z 316.236,A -85,B 0,C 180,E1 -31320,E2 -31320} C_VEL
LIN {X 0,Y 56.234,Z 316.66,A -85,B 0,C 180,E1 -31321.51,E2 -31321.51} C_VEL
LIN {X 0,Y 55.185,Z 317.739,A -85,B 0,C 180,E1 -31323.951,E2 -31323.951} C_VEL
LIN {X 0,Y 46.351,Z 323.374,A -85,B 0,C 180,E1 -31327.898,E2 -31327.898} C_VEL
LIN {X 0,Y 44.095,Z 324.648,A -85,B 0,C 180,E1 -31329.175,E2 -31329.175} C_VEL
LIN {X 0,Y 38.919,Z 327.105,A -85,B 0,C 180,E1 -31331.254,E2 -31331.254} C_VEL
LIN {X 0,Y 33.359,Z 329.11,A -85,B 0,C 180,E1 -31332.284,E2 -31332.284} C_VEL
LIN {X 0,Y 21.82,Z 332.107,A -85,B 0,C 180,E1 -31334.405,E2 -31334.405} C_VEL
LIN {X 0,Y 16.247,Z 333.15,A -85,B 0,C 180,E1 -31339.757,E2 -31339.757} C_VEL
LIN {X 0,Y 14.565,Z 333.426,A -85,B 0,C 180,E1 -31343.492,E2 -31343.492} C_VEL
LIN {X 0,Y 10.024,Z 334.255,A -85,B 0,C 180,E1 -31365.556,E2 -31365.556} C_VEL
LIN {X 0,Y 8.672,Z 334.718,A -85,B 0,C 180,E1 -31410.06,E2 -31410.06} C_VEL
LIN {X 0,Y 12.477,Z 334.664,A -85,B 0,C 180,E1 -31444.332,E2 -31444.332} C_VEL
LIN {X 0,Y 19.928,Z 333.902,A -85,B 0,C 180,E1 -31462.352,E2 -31462.352} C_VEL
LIN {X 0,Y 19.883,Z 333.252,A -85,B 0,C 180,E1 -31471.609,E2 -31471.609} C_VEL
LIN {X 0,Y 21.485,Z 330.306,A -85,B 0,C 180,E1 -31524.154,E2 -31524.154} C_VEL
LIN {X 0,Y 19.768,Z 330.604,A -85,B 0,C 180,E1 -31532.271,E2 -31532.271} C_VEL
LIN {X 0,Y 12.798,Z 331.755,A -85,B 0,C 180,E1 -31556.644,E2 -31556.644} C_VEL
LIN {X 0,Y 10.692,Z 332.034,A -85,B 0,C 180,E1 -31589.951,E2 -31589.951} C_VEL
LIN {X 0,Y 12.788,Z 331.781,A -85,B 0,C 180,E1 -31623.289,E2 -31623.289} C_VEL
LIN {X 0,Y 17.62,Z 331.075,A -85,B 0,C 180,E1 -31642.864,E2 -31642.864} C_VEL
LIN {X 0,Y 23.493,Z 329.857,A -85,B 0,C 180,E1 -31653.775,E2 -31653.775} C_VEL
LIN {X 0,Y 33.225,Z 327.044,A -85,B 0,C 180,E1 -31662.098,E2 -31662.098} C_VEL
LIN {X 0,Y 43.16,Z 323.006,A -85,B 0,C 180,E1 -31667.633,E2 -31667.633} C_VEL
LIN {X 0,Y 49.998,Z 319.473,A -85,B 0,C 180,E1 -31669.663,E2 -31669.663} C_VEL
LIN {X 0,Y 51.101,Z 318.928,A -85,B 0,C 180,E1 -31672.095,E2 -31672.095} C_VEL
LIN {X 0,Y 50.898,Z 319.238,A -85,B 0,C 180,E1 -31674.944,E2 -31674.944} C_VEL
LIN {X 0,Y 49.225,Z 320.465,A -85,B 0,C 180,E1 -31677.738,E2 -31677.738} C_VEL
LIN {X 0,Y 38.655,Z 325.963,A -85,B 0,C 180,E1 -31681.347,E2 -31681.347} C_VEL
LIN {X 0,Y 28.252,Z 329.942,A -85,B 0,C 180,E1 -31685.885,E2 -31685.885} C_VEL
LIN {X 0,Y 21.502,Z 331.888,A -85,B 0,C 180,E1 -31691.443,E2 -31691.443} C_VEL
LIN {X 0,Y 14.565,Z 333.426,A -85,B 0,C 180,E1 -31703.492,E2 -31703.492} C_VEL
LIN {X 0,Y 11.118,Z 333.916,A -85,B 0,C 180,E1 -31712.403,E2 -31712.403} C_VEL
LIN {X 0,Y 5.267,Z 334.083,A -85,B 0,C 180,E1 -31738.034,E2 -31738.034} C_VEL
LIN {X 0,Y 4.876,Z 333.853,A -85,B 0,C 180,E1 -31821.44,E2 -31821.44} C_VEL
LIN {X 0,Y 8.451,Z 333.635,A -85,B 0,C 180,E1 -31837.154,E2 -31837.154} C_VEL
LIN {X 0,Y 10.937,Z 333.488,A -85,B 0,C 180,E1 -31839.482,E2 -31839.482} C_VEL
LIN {X 0,Y 11.387,Z 333.093,A -85,B 0,C 180,E1 -31850.83,E2 -31850.83} C_VEL
LIN {X 0,Y 11.805,Z 332.541,A -85,B 0,C 180,E1 -31868.9,E2 -31868.9} C_VEL
LIN {X 0,Y 11.071,Z 332.427,A -85,B 0,C 180,E1 -31879.218,E2 -31879.218} C_VEL
LIN {X 0,Y 3.664,Z 333.008,A -85,B 0,C 180,E1 -31949.858,E2 -31949.858} C_VEL
LIN {X 0,Y 7.917,Z 332.755,A -85,B 0,C 180,E1 -32012.448,E2 -32012.448} C_VEL
LIN {X 0,Y 14.503,Z 332.049,A -85,B 0,C 180,E1 -32025.59,E2 -32025.59} C_VEL
LIN {X 0,Y 21.339,Z 330.832,A -85,B 0,C 180,E1 -32030.968,E2 -32030.968} C_VEL
LIN {X 0,Y 21.275,Z 330.892,A -85,B 0,C 180,E1 -32032.124,E2 -32032.124} C_VEL
LIN {X 0,Y 11.852,Z 332.63,A -85,B 0,C 180,E1 -32034.88,E2 -32034.88} C_VEL
LIN {X 0,Y 1.47,Z 333.72,A -85,B 0,C 180,E1 -32130.353,E2 -32130.353} C_VEL
LIN {X 0,Y 8.451,Z 333.635,A -85,B 0,C 180,E1 -32197.154,E2 -32197.154} C_VEL
LIN {X 0,Y 10.51,Z 335.633,A -85,B 0,C 180,E1 -32199.007,E2 -32199.007} C_VEL
LIN {X 0,Y 10.51,Z 600,A -85,B 0,C 180,E1 -32199.007,E2 -32199.007} C_VEL
LIN {X 0,Y 10.51,Z 600,A -85,B 0,C 180,E1 -32199.007,E2 -32199.007}

QRS_NEXT_CUT()

QRS_NEXT()
QRS_HOME()

END
